SUBAPPLICATION Uebung_040 (* Lauflicht 8 *)
  (* Standard: 61499-2; Description: Copyright (c) 2023 Meisterschulen am Ostbahnhof This program and the accompanying materials are made available under the terms of the Eclipse Public License 2.0 which is available at https://www.eclipse.org/legal/epl-2.0/ SPDX-License-Identifier: EPL-2.0 *)
  (* Version 1.0, 2023-10-23, Franz Höpfinger, Meisterschulen am Ostbahnhof, initial API and implementation and/or initial documentation *)
  PACKAGE Uebungen;
  IMPORT Uebungen::const::UT::DefaultPool::OutputNumber_N1;
  IMPORT logiBUS::io::DI::logiBUS_DI::Input_I1;
  IMPORT logiBUS::io::DI::logiBUS_DI::Input_I2;
  IMPORT logiBUS::io::DI::logiBUS_DI::Input_I3;
  IMPORT logiBUS::io::DI::logiBUS_DI::Input_I4;
  IMPORT logiBUS::io::DI::logiBUS_DI_Events::BUTTON_SINGLE_CLICK;
  IMPORT logiBUS::io::DQ::logiBUS_DO::Output_Q1;
  IMPORT logiBUS::io::DQ::logiBUS_DO::Output_Q2;
  IMPORT logiBUS::io::DQ::logiBUS_DO::Output_Q3;
  IMPORT logiBUS::io::DQ::logiBUS_DO::Output_Q4;
  IMPORT logiBUS::io::DQ::logiBUS_DO::Output_Q5;
  IMPORT logiBUS::io::DQ::logiBUS_DO::Output_Q6;
  IMPORT logiBUS::io::DQ::logiBUS_DO::Output_Q7;
  IMPORT logiBUS::io::DQ::logiBUS_DO::Output_Q8;
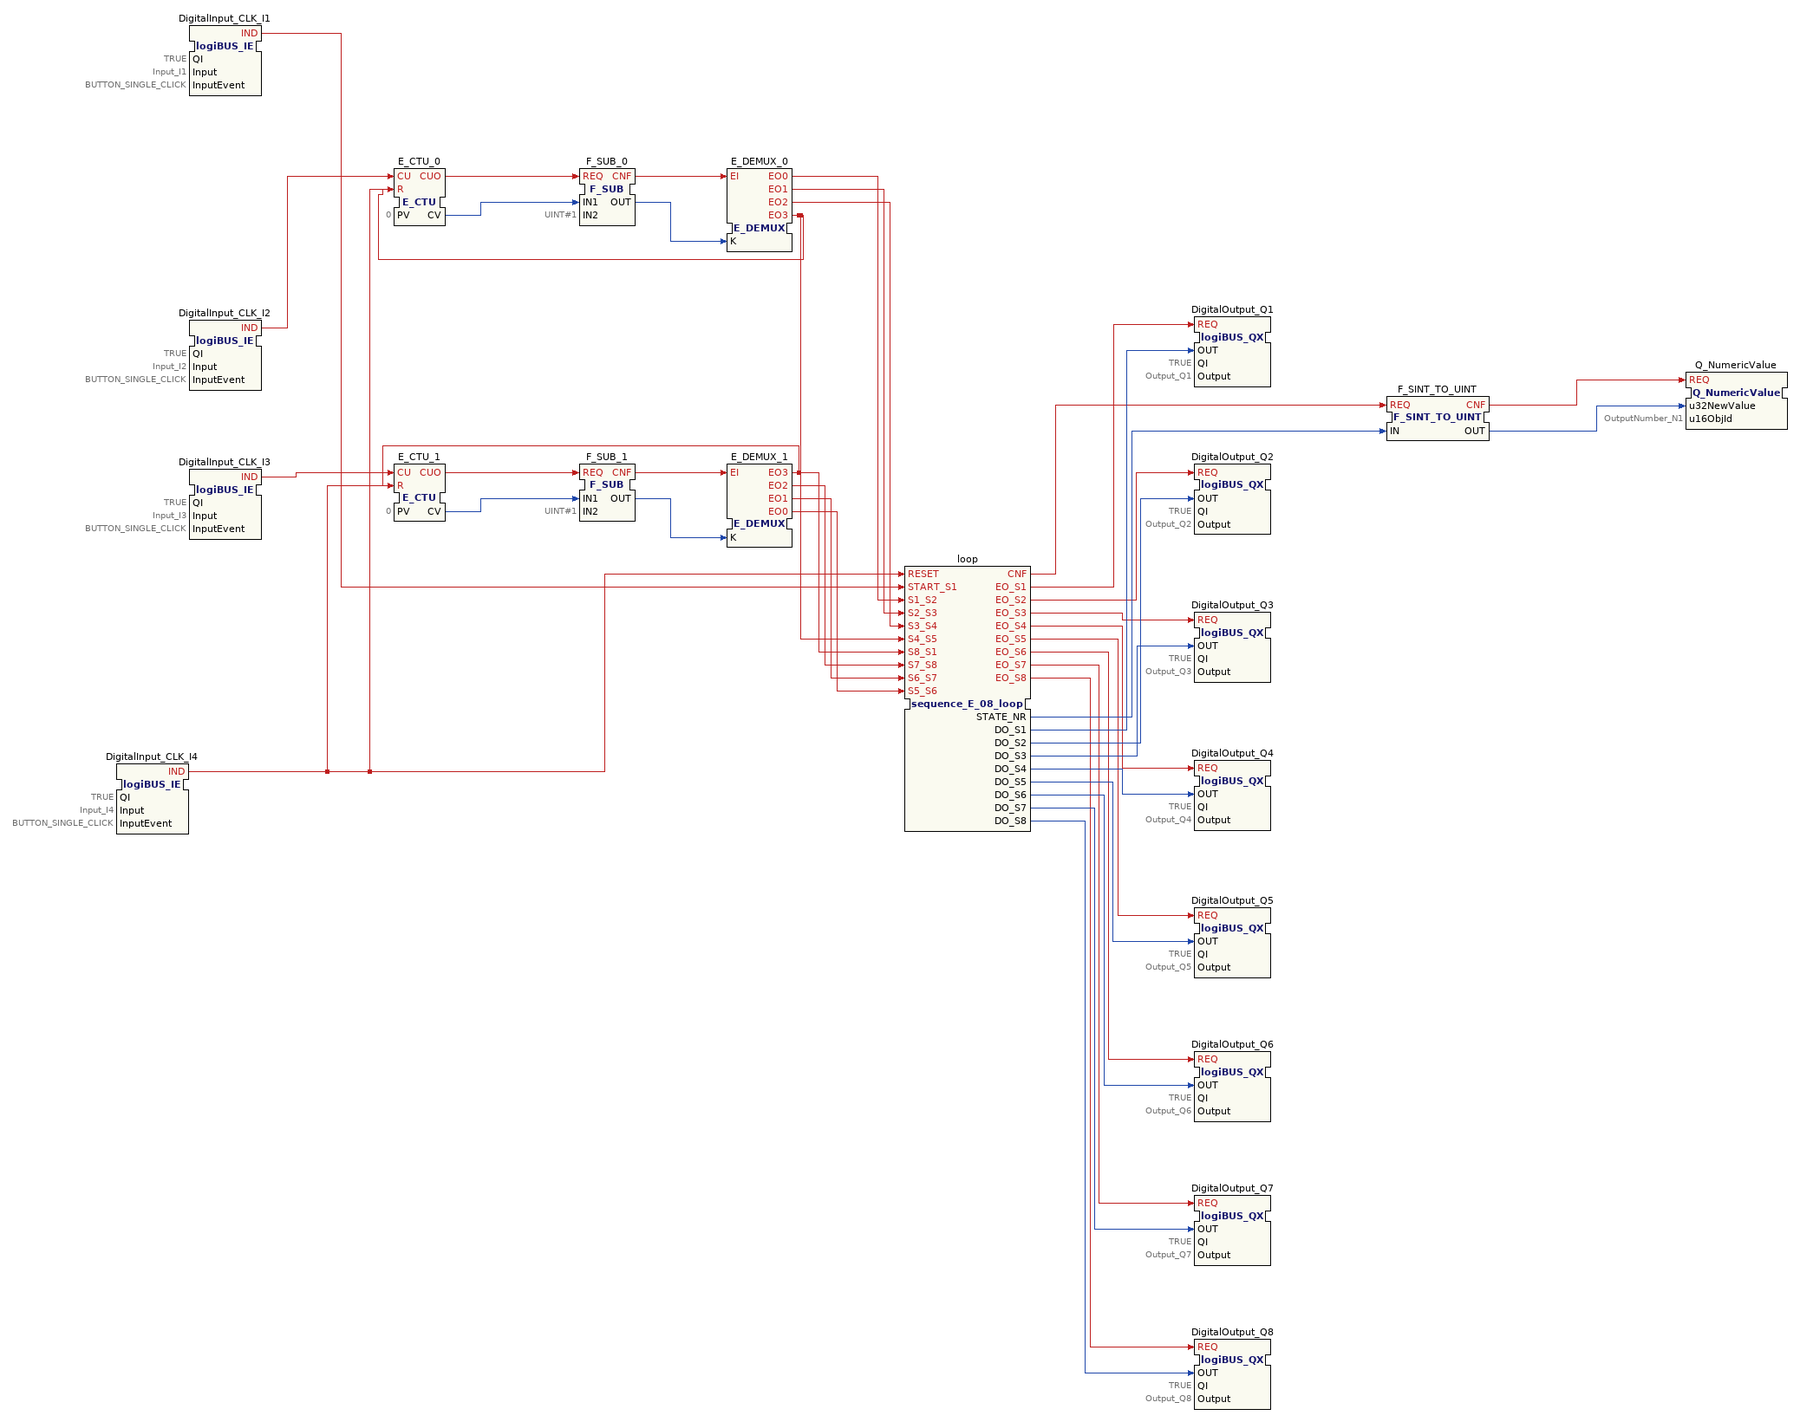
  FBS
    DigitalOutput_Q1 : logiBUS::io::DQ::logiBUS_QX(QI := TRUE, Output := Output_Q1);
    DigitalOutput_Q2 : logiBUS::io::DQ::logiBUS_QX(QI := TRUE, Output := Output_Q2);
    DigitalOutput_Q3 : logiBUS::io::DQ::logiBUS_QX(QI := TRUE, Output := Output_Q3);
    DigitalOutput_Q4 : logiBUS::io::DQ::logiBUS_QX(QI := TRUE, Output := Output_Q4);
    DigitalInput_CLK_I1 : logiBUS::io::DI::logiBUS_IE(QI := TRUE, Input := Input_I1, InputEvent := BUTTON_SINGLE_CLICK);
    DigitalInput_CLK_I4 : logiBUS::io::DI::logiBUS_IE(QI := TRUE, Input := Input_I4, InputEvent := BUTTON_SINGLE_CLICK);
    DigitalOutput_Q5 : logiBUS::io::DQ::logiBUS_QX(QI := TRUE, Output := Output_Q5);
    DigitalOutput_Q6 : logiBUS::io::DQ::logiBUS_QX(QI := TRUE, Output := Output_Q6);
    DigitalOutput_Q7 : logiBUS::io::DQ::logiBUS_QX(QI := TRUE, Output := Output_Q7);
    DigitalOutput_Q8 : logiBUS::io::DQ::logiBUS_QX(QI := TRUE, Output := Output_Q8);
    Q_NumericValue : isobus::UT::Q::Q_NumericValue(u16ObjId := OutputNumber_N1);
    F_SINT_TO_UINT : iec61131::conversion::F_SINT_TO_UINT;
    loop : logiBUS::utils::sequence::event::sequence_E_08_loop;
    E_CTU_0 : iec61499::events::E_CTU(PV := 0);
    E_DEMUX_0 : iec61499::events::E_DEMUX;
    DigitalInput_CLK_I2 : logiBUS::io::DI::logiBUS_IE(QI := TRUE, Input := Input_I2, InputEvent := BUTTON_SINGLE_CLICK);
    E_CTU_1 : iec61499::events::E_CTU(PV := 0);
    E_DEMUX_1 : iec61499::events::E_DEMUX;
    DigitalInput_CLK_I3 : logiBUS::io::DI::logiBUS_IE(QI := TRUE, Input := Input_I3, InputEvent := BUTTON_SINGLE_CLICK);
    F_SUB_1 : iec61131::arithmetic::F_SUB(IN2 := UINT#1);
    F_SUB_0 : iec61131::arithmetic::F_SUB(IN2 := UINT#1);
  END_FBS
  EVENT_CONNECTIONS
    F_SINT_TO_UINT.CNF TO Q_NumericValue.REQ;
    DigitalInput_CLK_I4.IND TO loop.RESET;
    loop.CNF TO F_SINT_TO_UINT.REQ;
    loop.EO_S1 TO DigitalOutput_Q1.REQ;
    loop.EO_S2 TO DigitalOutput_Q2.REQ;
    loop.EO_S3 TO DigitalOutput_Q3.REQ;
    loop.EO_S4 TO DigitalOutput_Q4.REQ;
    loop.EO_S5 TO DigitalOutput_Q5.REQ;
    loop.EO_S6 TO DigitalOutput_Q6.REQ;
    loop.EO_S7 TO DigitalOutput_Q7.REQ;
    loop.EO_S8 TO DigitalOutput_Q8.REQ;
    DigitalInput_CLK_I1.IND TO loop.START_S1;
    E_DEMUX_0.EO0 TO loop.S1_S2;
    E_DEMUX_0.EO1 TO loop.S2_S3;
    E_DEMUX_0.EO2 TO loop.S3_S4;
    E_DEMUX_0.EO3 TO loop.S4_S5;
    DigitalInput_CLK_I2.IND TO E_CTU_0.CU;
    DigitalInput_CLK_I3.IND TO E_CTU_1.CU;
    E_DEMUX_1.EO3 TO loop.S8_S1;
    E_DEMUX_1.EO2 TO loop.S7_S8;
    E_DEMUX_1.EO1 TO loop.S6_S7;
    E_DEMUX_1.EO0 TO loop.S5_S6;
    F_SUB_1.CNF TO E_DEMUX_1.EI;
    F_SUB_0.CNF TO E_DEMUX_0.EI;
    E_CTU_0.CUO TO F_SUB_0.REQ;
    E_CTU_1.CUO TO F_SUB_1.REQ;
    DigitalInput_CLK_I4.IND TO E_CTU_1.R;
    DigitalInput_CLK_I4.IND TO E_CTU_0.R;
    E_DEMUX_0.EO3 TO E_CTU_0.R;
    E_DEMUX_1.EO3 TO E_CTU_1.R;
  END_CONNECTIONS
  DATA_CONNECTIONS
    F_SINT_TO_UINT.OUT TO Q_NumericValue.u32NewValue;
    loop.STATE_NR TO F_SINT_TO_UINT.IN;
    loop.DO_S1 TO DigitalOutput_Q1.OUT;
    loop.DO_S2 TO DigitalOutput_Q2.OUT;
    loop.DO_S3 TO DigitalOutput_Q3.OUT;
    loop.DO_S4 TO DigitalOutput_Q4.OUT;
    loop.DO_S5 TO DigitalOutput_Q5.OUT;
    loop.DO_S6 TO DigitalOutput_Q6.OUT;
    loop.DO_S7 TO DigitalOutput_Q7.OUT;
    loop.DO_S8 TO DigitalOutput_Q8.OUT;
    F_SUB_1.OUT TO E_DEMUX_1.K;
    F_SUB_0.OUT TO E_DEMUX_0.K;
    E_CTU_0.CV TO F_SUB_0.IN1;
    E_CTU_1.CV TO F_SUB_1.IN1;
  END_CONNECTIONS
END_SUBAPPLICATION
